KUKA KRL program: wkz1_ok.src, wkz1_ok.dat

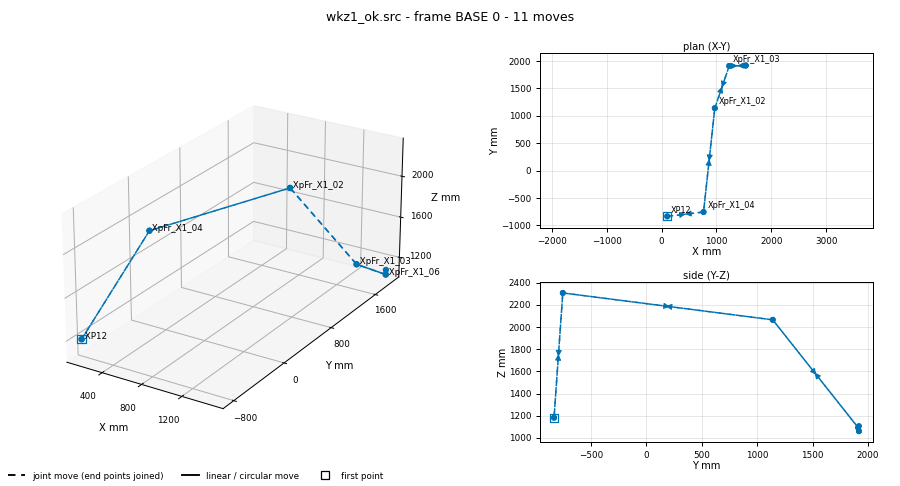
[picture p0: tool path of wkz1_ok.src in frame BASE 0, 11 of 11 moves have a stored position in this frame; points joined in program order, loops and branches not executed]
--- wkz1_ok.src ---
&ACCESS RVP
&REL 1
&COMMENT CHECK TCP X1
&PARAM DISKPATH = KRC:\R1\Program
&PARAM TEMPLATE = C:\KRC\Roboter\Template\vorgabe
&PARAM EDITMASK = *
DEF wkz1_ok( )
;FOLD INI
  ;FOLD BASISTECH INI
    GLOBAL INTERRUPT DECL 3 WHEN $STOPMESS==TRUE DO IR_STOPM ( )
    INTERRUPT ON 3
    BAS (#INITMOV,0 )
  ;ENDFOLD (BASISTECH INI)
;FOLD SPOTTECH INI
USERSPOT(#INIT)
;ENDFOLD (SPOTTECH INI)
;FOLD GRIPPERTECH INI
USER_GRP(0,DUMMY,DUMMY,GDEFAULT)
;ENDFOLD (GRIPPERTECH INI)
  ;FOLD USER INI
    ;Make your modifications here

  ;ENDFOLD (USER INI)
;ENDFOLD (INI)

; Caracterização dos meios de produção:
; CHANGES: Check TCP GUN X1
; Versão Atual:08/10/2015
; Name: P13.050-R1

chk_w1_wechs_ok ( )              ; CHECK X1

;FOLD PTP P12 Vel=100 % PDAT12 Tool[1]:GUN X1 Base[0];%{PE}%R 8.2.20,%MKUKATPBASIS,%CMOVE,%VPTP,%P 1:PTP, 2:P12, 3:, 5:100, 7:PDAT12
$BWDSTART=FALSE
PDAT_ACT=PPDAT12
FDAT_ACT=FP12
BAS(#PTP_PARAMS,100)
PTP XP12
;ENDFOLD
;FOLD PTP pFr_X1_04 CONT Vel=100 % PDAT13 Tool[1]:GUN X1 Base[0];%{PE}%R 8.2.20,%MKUKATPBASIS,%CMOVE,%VPTP,%P 1:PTP, 2:pFr_X1_04, 3:C_DIS, 5:100, 7:PDAT13
$BWDSTART=FALSE
PDAT_ACT=PPDAT13
FDAT_ACT=FpFr_X1_04
BAS(#PTP_PARAMS,100)
PTP XpFr_X1_04 C_DIS
;ENDFOLD
;FOLD PTP pFr_X1_02 CONT Vel=100 % PDAT14 Tool[1]:GUN X1 Base[0];%{PE}%R 8.2.20,%MKUKATPBASIS,%CMOVE,%VPTP,%P 1:PTP, 2:pFr_X1_02, 3:C_DIS, 5:100, 7:PDAT14
$BWDSTART=FALSE
PDAT_ACT=PPDAT14
FDAT_ACT=FpFr_X1_02
BAS(#PTP_PARAMS,100)
PTP XpFr_X1_02 C_DIS
;ENDFOLD
;FOLD PTP pFr_X1_03 CONT Vel=100 % PDAT15 Tool[1]:GUN X1 Base[0];%{PE}%R 8.2.20,%MKUKATPBASIS,%CMOVE,%VPTP,%P 1:PTP, 2:pFr_X1_03, 3:C_DIS, 5:100, 7:PDAT15
$BWDSTART=FALSE
PDAT_ACT=PPDAT15
FDAT_ACT=FpFr_X1_03
BAS(#PTP_PARAMS,100)
PTP XpFr_X1_03 C_DIS
;ENDFOLD
;FOLD LIN pFr_X1_06 Vel=0.25 m/s CPDAT0 Tool[1]:GUN X1 Base[0];%{PE}%R 8.2.20,%MKUKATPBASIS,%CMOVE,%VLIN,%P 1:LIN, 2:pFr_X1_06, 3:, 5:0.25, 7:CPDAT0
$BWDSTART=FALSE
LDAT_ACT=LCPDAT0
FDAT_ACT=FpFr_X1_06
BAS(#CP_PARAMS,0.25)
LIN XpFr_X1_06
;ENDFOLD

;FOLD ; POSICAO CHECK X1;%{PE}%R 8.2.20,%MKUKATPBASIS,%CCOMMENT,%VNORMAL,%P 2:POSICAO  CHECK  X1
;ENDFOLD
;FOLD LIN pFr_X1_08 CONT Vel=0.2 m/s CPDAT4 Tool[1]:GUN X1 Base[0];%{PE}%R 8.2.20,%MKUKATPBASIS,%CMOVE,%VLIN,%P 1:LIN, 2:pFr_X1_08, 3:C_DIS C_DIS, 5:0.2, 7:CPDAT4
$BWDSTART=FALSE
LDAT_ACT=LCPDAT4
FDAT_ACT=FpFr_X1_08
BAS(#CP_PARAMS,0.2)
LIN XpFr_X1_08 C_DIS C_DIS
;ENDFOLD
;FOLD WAIT Time=5 sec;%{PE}%R 8.2.20,%MKUKATPBASIS,%CWAIT,%VWAIT,%P 3:5
WAIT SEC 5
;ENDFOLD

;FOLD LIN pFr_X1_09 CONT Vel=0.35 m/s CPDAT5 Tool[1]:GUN X1 Base[0];%{PE}%R 8.2.20,%MKUKATPBASIS,%CMOVE,%VLIN,%P 1:LIN, 2:pFr_X1_09, 3:C_DIS C_DIS, 5:0.35, 7:CPDAT5
$BWDSTART=FALSE
LDAT_ACT=LCPDAT5
FDAT_ACT=FpFr_X1_09
BAS(#CP_PARAMS,0.35)
LIN XpFr_X1_09 C_DIS C_DIS
;ENDFOLD
;FOLD PTP pFr_X1_11 CONT Vel=100 % PDAT19 Tool[1]:GUN X1 Base[0];%{PE}%R 8.2.20,%MKUKATPBASIS,%CMOVE,%VPTP,%P 1:PTP, 2:pFr_X1_11, 3:C_DIS, 5:100, 7:PDAT19
$BWDSTART=FALSE
PDAT_ACT=PPDAT19
FDAT_ACT=FpFr_X1_11
BAS(#PTP_PARAMS,100)
PTP XpFr_X1_11 C_DIS
;ENDFOLD
;FOLD PTP pFr_X1_12 CONT Vel=100 % PDAT20 Tool[1]:GUN X1 Base[0];%{PE}%R 8.2.20,%MKUKATPBASIS,%CMOVE,%VPTP,%P 1:PTP, 2:pFr_X1_12, 3:C_DIS, 5:100, 7:PDAT20
$BWDSTART=FALSE
PDAT_ACT=PPDAT20
FDAT_ACT=FpFr_X1_12
BAS(#PTP_PARAMS,100)
PTP XpFr_X1_12 C_DIS
;ENDFOLD
;FOLD PTP pFr_X1_07 CONT Vel=100 % PDAT21 Tool[1]:GUN X1 Base[0];%{PE}%R 8.2.20,%MKUKATPBASIS,%CMOVE,%VPTP,%P 1:PTP, 2:pFr_X1_07, 3:C_DIS, 5:100, 7:PDAT21
$BWDSTART=FALSE
PDAT_ACT=PPDAT21
FDAT_ACT=FpFr_X1_07
BAS(#PTP_PARAMS,100)
PTP XpFr_X1_07 C_DIS
;ENDFOLD
;FOLD PTP P14 Vel=100 % PDAT22 Tool[1]:GUN X1 Base[0];%{PE}%R 8.2.20,%MKUKATPBASIS,%CMOVE,%VPTP,%P 1:PTP, 2:P14, 3:, 5:100, 7:PDAT22
$BWDSTART=FALSE
PDAT_ACT=PPDAT22
FDAT_ACT=FP14
BAS(#PTP_PARAMS,100)
PTP XP14
;ENDFOLD

END

--- wkz1_ok.dat ---
&ACCESS RVP
&REL 1
&COMMENT CHECK TCP X1
&PARAM DISKPATH = KRC:\R1\Program
&PARAM TEMPLATE = C:\KRC\Roboter\Template\vorgabe
&PARAM EDITMASK = *
DEFDAT wkz1_ok
;FOLD EXTERNAL DECLARATIONS;%{PE}%MKUKATPBASIS,%CEXT,%VCOMMON,%P
;FOLD GRIPPERTECH EXT
EXT  H50 (INT  :IN,INT  :IN,INT  :IN,GRP_TYP  :IN )
;ENDFOLD (GRIPPERTECH EXT)
;FOLD SPOTTECH EXT
EXT  USERSPOT (S_COMMAND  :IN,SPOT_TYPE  :IN )
;ENDFOLD (SPOTTECH EXT)
;FOLD BASISTECH EXT;%{PE}%MKUKATPBASIS,%CEXT,%VEXT,%P
EXT  BAS (BAS_COMMAND  :IN,REAL  :IN )
DECL INT SUCCESS
;ENDFOLD (BASISTECH EXT)
;FOLD USER EXT;%{E}%MKUKATPUSER,%CEXT,%VEXT,%P
;Make your modifications here

;ENDFOLD (USER EXT)
;ENDFOLD (EXTERNAL DECLARATIONS)
DECL BASIS_SUGG_T LAST_BASIS={POINT1[] "P14                     ",POINT2[] "P14                     ",CP_PARAMS[] "CPDAT5                  ",PTP_PARAMS[] "PDAT22                  ",CONT[] "                        ",CP_VEL[] "0.35                    ",PTP_VEL[] "25                      ",SYNC_PARAMS[] "SYNCDAT                 ",SPL_NAME[] "S0                      "}
DECL E6POS XP1={X 41.948761,Y 1188.81604,Z 963.694824,A 98.9483032,B 81.6207123,C 97.2233963,S 2,T 11,E1 213.504807,E2 0.0,E3 0.0,E4 0.0,E5 0.0,E6 0.0}
DECL FDAT FP1={TOOL_NO 1,BASE_NO 0,IPO_FRAME #BASE,POINT2[] " ",TQ_STATE FALSE}
DECL PDAT PPDAT1={VEL 100.0,ACC 100.0,APO_DIST 100.0,APO_MODE #CDIS}
DECL E6POS XP2={X -877.220825,Y 739.940186,Z 1288.67004,A 173.423203,B 23.5768509,C -178.225296,S 2,T 11,E1 -1009.36298,E2 0.0,E3 0.0,E4 0.0,E5 0.0,E6 0.0}
DECL FDAT FP2={TOOL_NO 1,BASE_NO 0,IPO_FRAME #BASE,POINT2[] " ",TQ_STATE FALSE}
DECL PDAT PPDAT2={VEL 100.0,ACC 100.0,APO_DIST 100.0,APO_MODE #CDIS}
DECL E6POS XP3={X -932.592224,Y 276.203491,Z 1065.61096,A 177.576004,B -2.90737295,C -177.044006,S 2,T 11,E1 -2111.32007,E2 0.0,E3 0.0,E4 0.0,E5 0.0,E6 0.0}
DECL FDAT FP3={TOOL_NO 1,BASE_NO 0,IPO_FRAME #BASE,POINT2[] " ",TQ_STATE FALSE}
DECL E6POS XP6={X -933.703491,Y 275.964386,Z 1031.41101,A 177.576004,B -2.90736103,C -177.044006,S 2,T 11,E1 -2111.32007,E2 0.0,E3 0.0,E4 0.0,E5 0.0,E6 0.0}
DECL FDAT FP6={TOOL_NO 1,BASE_NO 0,IPO_FRAME #BASE,POINT2[] " ",TQ_STATE FALSE}
DECL E6POS XP7={X -932.592224,Y 276.203491,Z 1065.61096,A 177.576004,B -2.90737295,C -177.044006,S 2,T 11,E1 -2111.32007,E2 0.0,E3 0.0,E4 0.0,E5 0.0,E6 0.0}
DECL FDAT FP7={TOOL_NO 1,BASE_NO 0,IPO_FRAME #BASE,POINT2[] " ",TQ_STATE FALSE}
DECL PDAT PPDAT8={VEL 100.0,ACC 100.0,APO_DIST 100.0,APO_MODE #CDIS}
DECL E6POS XP8={X -877.220825,Y 739.940186,Z 1288.67004,A 173.423203,B 23.5768509,C -178.225296,S 2,T 11,E1 -1009.36298,E2 0.0,E3 0.0,E4 0.0,E5 0.0,E6 0.0}
DECL FDAT FP8={TOOL_NO 1,BASE_NO 0,IPO_FRAME #BASE,POINT2[] " ",TQ_STATE FALSE}
DECL PDAT PPDAT11={VEL 100.0,ACC 100.0,APO_DIST 100.0,APO_MODE #CDIS}
DECL E6POS XP11={X 41.9489212,Y 1188.81604,Z 963.694885,A 98.9482498,B 81.620697,C 97.2233582,S 2,T 11,E1 213.504898,E2 0.0,E3 0.0,E4 0.0,E5 0.0,E6 0.0}
DECL FDAT FP11={TOOL_NO 1,BASE_NO 0,IPO_FRAME #BASE,POINT2[] " ",TQ_STATE FALSE}
DECL LDAT LCPDAT1={VEL 2.0,ACC 100.0,APO_DIST 100.0,APO_FAC 50.0,AXIS_VEL 100.0,AXIS_ACC 100.0,ORI_TYP #VAR,CIRC_TYP #BASE,JERK_FAC 50.0,GEAR_JERK 50.0,EXAX_IGN 0}
DECL LDAT LCPDAT2={VEL 2.0,ACC 100.0,APO_DIST 100.0,APO_FAC 50.0,AXIS_VEL 100.0,AXIS_ACC 100.0,ORI_TYP #VAR,CIRC_TYP #BASE,JERK_FAC 50.0,GEAR_JERK 50.0,EXAX_IGN 0}
DECL LDAT LCPDAT3={VEL 2.0,ACC 100.0,APO_DIST 100.0,APO_FAC 50.0,AXIS_VEL 100.0,AXIS_ACC 100.0,ORI_TYP #VAR,CIRC_TYP #BASE,JERK_FAC 50.0,GEAR_JERK 50.0,EXAX_IGN 0}
DECL PDAT PPDAT12={VEL 100.0,ACC 100.0,APO_DIST 100.0,APO_MODE #CDIS}
DECL E6POS XP12={X 101.904198,Y -833.887207,Z 1182.97998,A -87.0955505,B 79.0952911,C 80.3321075,S 2,T 2,E1 213.625793,E2 0.0,E3 0.0,E4 0.0,E5 0.0,E6 0.0}
DECL FDAT FP12={TOOL_NO 1,BASE_NO 0,IPO_FRAME #BASE,POINT2[] " ",TQ_STATE FALSE}
DECL PDAT PPDAT13={VEL 100.0,ACC 100.0,APO_DIST 100.0,APO_MODE #CDIS}
DECL E6POS XpFr_X1_04={X 763.830505,Y -754.804016,Z 2308.69702,A -54.2272797,B 44.6665993,C 55.8185196,S 2,T 3,E1 207.1996,E2 0.0,E3 0.0,E4 0.0,E5 0.0,E6 0.0}
DECL FDAT FpFr_X1_04={TOOL_NO 1,BASE_NO 0,IPO_FRAME #BASE,POINT2[] " ",TQ_STATE FALSE}
DECL PDAT PPDAT14={VEL 100.0,ACC 100.0,APO_DIST 100.0,APO_MODE #CDIS}
DECL E6POS XpFr_X1_02={X 969.039673,Y 1139.73096,Z 2066.15308,A 44.3954697,B 54.7452507,C 92.8609467,S 2,T 3,E1 199.989594,E2 0.0,E3 0.0,E4 0.0,E5 0.0,E6 0.0}
DECL FDAT FpFr_X1_02={TOOL_NO 1,BASE_NO 0,IPO_FRAME #BASE,POINT2[] " ",TQ_STATE FALSE}
DECL PDAT PPDAT15={VEL 100.0,ACC 100.0,APO_DIST 100.0,APO_MODE #CDIS}
DECL E6POS XpFr_X1_03={X 1232.01599,Y 1909.97595,Z 1094.03296,A 0.817309082,B 6.79582977,C -0.246864095,S 2,T 35,E1 -532.459717,E2 0.0,E3 0.0,E4 0.0,E5 0.0,E6 0.0}
DECL FDAT FpFr_X1_03={TOOL_NO 1,BASE_NO 0,IPO_FRAME #BASE,POINT2[] " ",TQ_STATE FALSE}
DECL PDAT PPDAT16={VEL 100.0,ACC 100.0,APO_DIST 100.0,APO_MODE #CDIS}
DECL E6POS XpFr_X1_05={X 1286.05005,Y 1686.81702,Z 755.587097,A 0.624875784,B 1.75245798,C 1.14266706,S 2,T 35,E1 -532.457886,E2 0.0,E3 0.0,E4 0.0,E5 0.0,E6 0.0}
DECL FDAT FpFr_X1_05={TOOL_NO 1,BASE_NO 0,IPO_FRAME #BASE,POINT2[] " ",TQ_STATE FALSE}
DECL LDAT LCPDAT0={VEL 2.0,ACC 100.0,APO_DIST 100.0,APO_FAC 50.0,AXIS_VEL 100.0,AXIS_ACC 100.0,ORI_TYP #VAR,CIRC_TYP #BASE,JERK_FAC 50.0,GEAR_JERK 50.0,EXAX_IGN 0}
DECL E6POS XpFr_X1_06={X 1533.64001,Y 1917.64294,Z 1061.04504,A 0.817309201,B 6.79583216,C -0.2468642,S 2,T 35,E1 -532.460205,E2 0.0,E3 0.0,E4 0.0,E5 0.0,E6 0.0}
DECL FDAT FpFr_X1_06={TOOL_NO 1,BASE_NO 0,IPO_FRAME #BASE,POINT2[] " ",TQ_STATE FALSE}
DECL LDAT LCPDAT4={VEL 2.0,ACC 100.0,APO_DIST 100.0,APO_FAC 50.0,AXIS_VEL 100.0,AXIS_ACC 100.0,ORI_TYP #VAR,CIRC_TYP #BASE,JERK_FAC 50.0,GEAR_JERK 50.0,EXAX_IGN 0}
DECL E6POS XpFr_X1_08={X 1533.64001,Y 1917.64294,Z 1107.61499,A 0.817309201,B 6.79583216,C -0.2468642,S 2,T 35,E1 -532.460205,E2 0.0,E3 0.0,E4 0.0,E5 0.0,E6 0.0}
DECL FDAT FpFr_X1_08={TOOL_NO 1,BASE_NO 0,IPO_FRAME #BASE,POINT2[] " ",TQ_STATE FALSE}
DECL LDAT LCPDAT5={VEL 2.0,ACC 100.0,APO_DIST 100.0,APO_FAC 50.0,AXIS_VEL 100.0,AXIS_ACC 100.0,ORI_TYP #VAR,CIRC_TYP #BASE,JERK_FAC 50.0,GEAR_JERK 50.0,EXAX_IGN 0}
DECL E6POS XpFr_X1_09={X 1533.64001,Y 1917.64294,Z 1061.04504,A 0.817309201,B 6.79583216,C -0.2468642,S 2,T 35,E1 -532.460205,E2 0.0,E3 0.0,E4 0.0,E5 0.0,E6 0.0}
DECL FDAT FpFr_X1_09={TOOL_NO 1,BASE_NO 0,IPO_FRAME #BASE,POINT2[] " ",TQ_STATE FALSE}
DECL SPOT_SUGG_T LAST_SPOT={GUN[] " 1                      ",RETR_CMD[] "#OPN                    ",CHOISE[] "#FIRST                  ",CLO_TM[] "0                       ",PGNO1[] " 1                      ",PRESS1[] "0                       ",PGNO2[] " 1                      ",PRESS2[] "0                       ",SPOT_PARAMS[] "NORMAL                  "}
DECL PDAT PPDAT17={VEL 100.0,ACC 100.0,APO_DIST 100.0,APO_MODE #CDIS}
DECL E6POS XP13={X 9762.19434,Y -3811.4519,Z -756.436829,A -89.2618332,B 22.6249809,C -0.268216789,S 2,T 35,E1 -532.459717,E2 0.0,E3 0.0,E4 0.0,E5 0.0,E6 0.0}
DECL FDAT FP13={TOOL_NO 1,BASE_NO 1,IPO_FRAME #BASE,POINT2[] " ",TQ_STATE FALSE}
DECL PDAT PPDAT18={VEL 100.0,ACC 100.0,APO_DIST 100.0,APO_MODE #CDIS}
DECL E6POS XpFr_X1_10={X 1003.46301,Y 1260.20398,Z 880.076172,A 5.04273415,B 32.9262886,C 2.90043402,S 2,T 35,E1 -382.985596,E2 0.0,E3 0.0,E4 0.0,E5 0.0,E6 0.0}
DECL FDAT FpFr_X1_10={TOOL_NO 1,BASE_NO 0,IPO_FRAME #BASE,POINT2[] " ",TQ_STATE FALSE}
DECL PDAT PPDAT19={VEL 100.0,ACC 100.0,APO_DIST 100.0,APO_MODE #CDIS}
DECL E6POS XpFr_X1_11={X 1232.01599,Y 1909.97595,Z 1094.03296,A 0.817309082,B 6.79582977,C -0.246864095,S 2,T 35,E1 -532.459717,E2 0.0,E3 0.0,E4 0.0,E5 0.0,E6 0.0}
DECL FDAT FpFr_X1_11={TOOL_NO 1,BASE_NO 0,IPO_FRAME #BASE,POINT2[] " ",TQ_STATE FALSE}
DECL PDAT PPDAT20={VEL 100.0,ACC 100.0,APO_DIST 100.0,APO_MODE #CDIS}
DECL E6POS XpFr_X1_12={X 969.039673,Y 1139.73096,Z 2066.15308,A 44.3954697,B 54.7452507,C 92.8609467,S 2,T 3,E1 199.989594,E2 0.0,E3 0.0,E4 0.0,E5 0.0,E6 0.0}
DECL FDAT FpFr_X1_12={TOOL_NO 1,BASE_NO 0,IPO_FRAME #BASE,POINT2[] " ",TQ_STATE FALSE}
DECL PDAT PPDAT21={VEL 100.0,ACC 100.0,APO_DIST 100.0,APO_MODE #CDIS}
DECL E6POS XpFr_X1_07={X 763.830505,Y -754.804016,Z 2308.69702,A -54.2272797,B 44.6665993,C 55.8185196,S 2,T 3,E1 207.1996,E2 0.0,E3 0.0,E4 0.0,E5 0.0,E6 0.0}
DECL FDAT FpFr_X1_07={TOOL_NO 1,BASE_NO 0,IPO_FRAME #BASE,POINT2[] " ",TQ_STATE FALSE}
DECL PDAT PPDAT22={VEL 100.0,ACC 100.0,APO_DIST 100.0,APO_MODE #CDIS}
DECL E6POS XP14={X 101.904198,Y -833.887207,Z 1182.97998,A -87.0955505,B 79.0952911,C 80.3321075,S 2,T 2,E1 213.625793,E2 0.0,E3 0.0,E4 0.0,E5 0.0,E6 0.0}
DECL FDAT FP14={TOOL_NO 1,BASE_NO 0,IPO_FRAME #BASE,POINT2[] " ",TQ_STATE FALSE}
ENDDAT
